Fanuc KAREL source: webkee.kl

PROGRAM webkee
%COMMENT = 'legacy v1'
%NOLOCKGROUP
%NOPAUSE=ERROR+COMMAND+TPENABLE
%NOBUSYLAMP

CONST

	R_WEBKEEP = 42

VAR

	STATUS: INTEGER
	return_code: INTEGER

BEGIN

	SET_REAL_REG(R_WEBKEEP, 0, STATUS)
	return_code = 204

END webkee
